FUNCTION_BLOCK SimplePiston
VAR_INPUT
	bEnable : BOOL;
END_VAR
VAR_OUTPUT
	busy : BOOL;
END_VAR
VAR
	pistonExtend AT %Q* : BOOL;
	pistonRetract AT %Q* : BOOL;
	
	extended AT %I* : BOOL;
	retracted AT %I* : BOOL;
	
	mode : (HOLD, IN, OUT);
END_VAR

IF
	NOT bEnable OR
	(retracted AND_THEN (pistonRetract OR mode = OUT)) OR
	(extended AND_THEN (pistonExtend OR mode = IN))
THEN
	mode := HOLD;
END_IF

CASE mode OF
	HOLD:
		pistonRetract := FALSE;
		pistonExtend := FALSE;
		
	IN:
		pistonRetract := FALSE;
		pistonExtend := TRUE;
	
	OUT:
		pistonRetract := TRUE;
		pistonExtend := FALSE;
	
END_CASE

busy := mode <> HOLD;

METHOD extend : BOOL
VAR_INPUT
END_VAR
mode := IN;
END_METHOD

METHOD retract : BOOL
VAR_INPUT
END_VAR
mode := OUT;

retract := retracted;
END_METHOD

METHOD stop : BOOL
VAR_INPUT
END_VAR
pistonExtend := FALSE;
pistonRetract := FALSE;
mode := HOLD;
END_METHOD

END_FUNCTION_BLOCK

(* stored: Version 1.1.0.1, ProductVersion 3.1.4024.11
   POU SimplePiston: Id {0b7d1323-ab3c-4527-8947-07c900a0019d}, SpecialFunc None
   Method extend: Id {1445913b-ea25-4077-a571-d047dfa08814}
   Method retract: Id {4caa366f-5640-4a48-acfd-50fd41a5c7d8}
   Method stop: Id {538ae10f-48c1-4d70-9b3c-2da92f3346c7} *)
